FUNCTION_BLOCK DINT_TO_COLOR
VAR_INPUT
	ENTRADA: DINT;
END_VAR
VAR_OUTPUT
	SALIDA: COLOR;
END_VAR
VAR

END_VAR

CASE ENTRADA OF
	2:
	SALIDA := AZUL;
	
	5:
	SALIDA := VERDE;
	
	8:
	SALIDA := METAL;
END_CASE

END_FUNCTION_BLOCK

(* stored: Version 1.1.0.1, ProductVersion 3.1.4024.12
   POU DINT_TO_COLOR: Id {277e2afd-88e6-46fa-8472-6536bd28b295}, SpecialFunc None *)
